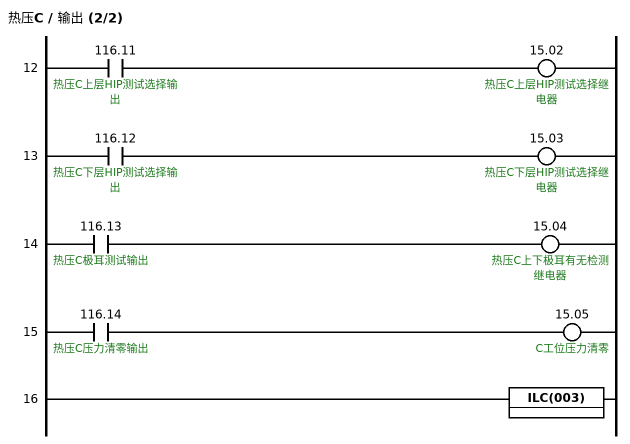
; rung 12
LD 116.11  ; 热压C上层HIP测试选择输出
OUT 15.02  ; 热压C上层HIP测试选择继电器
; rung 13
LD 116.12  ; 热压C下层HIP测试选择输出
OUT 15.03  ; 热压C下层HIP测试选择继电器
; rung 14
LD 116.13  ; 热压C极耳测试输出
OUT 15.04  ; 热压C上下极耳有无检测继电器
; rung 15
LD 116.14  ; 热压C压力清零输出
OUT 15.05  ; C工位压力清零
; rung 16
ILC(003)

### Section END
; rung 0
END(001)

## Program COM (cyclic task 7)

### Section 延时

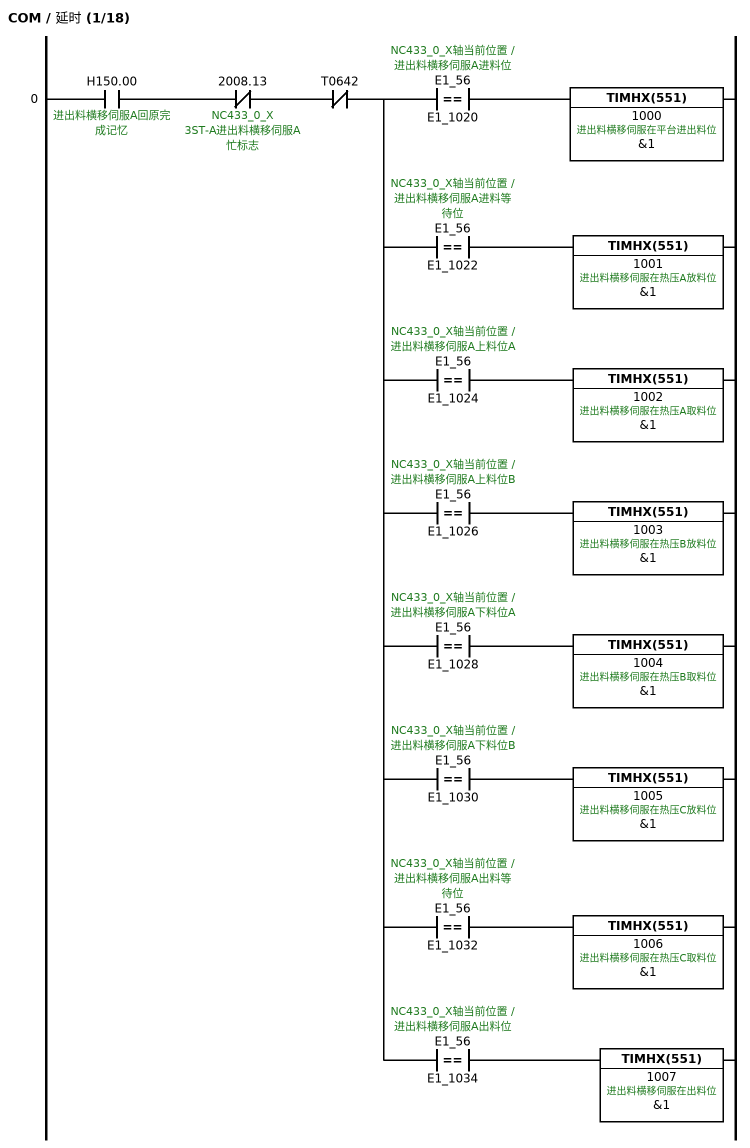
; rung 0
LD H150.00  ; 进出料横移伺服A回原完成记忆
ANDNOT 2008.13  ; NC433_0_X 3ST-A进出料横移伺服A忙标志
ANDNOT T0642
OUT TR0
AND=SL(303) E1_56 E1_1020  ; NC433_0_X轴当前位置, 进出料横移伺服A进料位
TIMHX(551) 1000 &1  ; 进出料横移伺服在平台进出料位
LD TR0
AND=SL(303) E1_56 E1_1022  ; NC433_0_X轴当前位置, 进出料横移伺服A进料等待位
TIMHX(551) 1001 &1  ; 进出料横移伺服在热压A放料位
LD TR0
AND=SL(303) E1_56 E1_1024  ; NC433_0_X轴当前位置, 进出料横移伺服A上料位A
TIMHX(551) 1002 &1  ; 进出料横移伺服在热压A取料位
LD TR0
AND=SL(303) E1_56 E1_1026  ; NC433_0_X轴当前位置, 进出料横移伺服A上料位B
TIMHX(551) 1003 &1  ; 进出料横移伺服在热压B放料位
LD TR0
AND=SL(303) E1_56 E1_1028  ; NC433_0_X轴当前位置, 进出料横移伺服A下料位A
TIMHX(551) 1004 &1  ; 进出料横移伺服在热压B取料位
LD TR0
AND=SL(303) E1_56 E1_1030  ; NC433_0_X轴当前位置, 进出料横移伺服A下料位B
TIMHX(551) 1005 &1  ; 进出料横移伺服在热压C放料位
LD TR0
AND=SL(303) E1_56 E1_1032  ; NC433_0_X轴当前位置, 进出料横移伺服A出料等待位
TIMHX(551) 1006 &1  ; 进出料横移伺服在热压C取料位
LD TR0
AND=SL(303) E1_56 E1_1034  ; NC433_0_X轴当前位置, 进出料横移伺服A出料位
TIMHX(551) 1007 &1  ; 进出料横移伺服在出料位

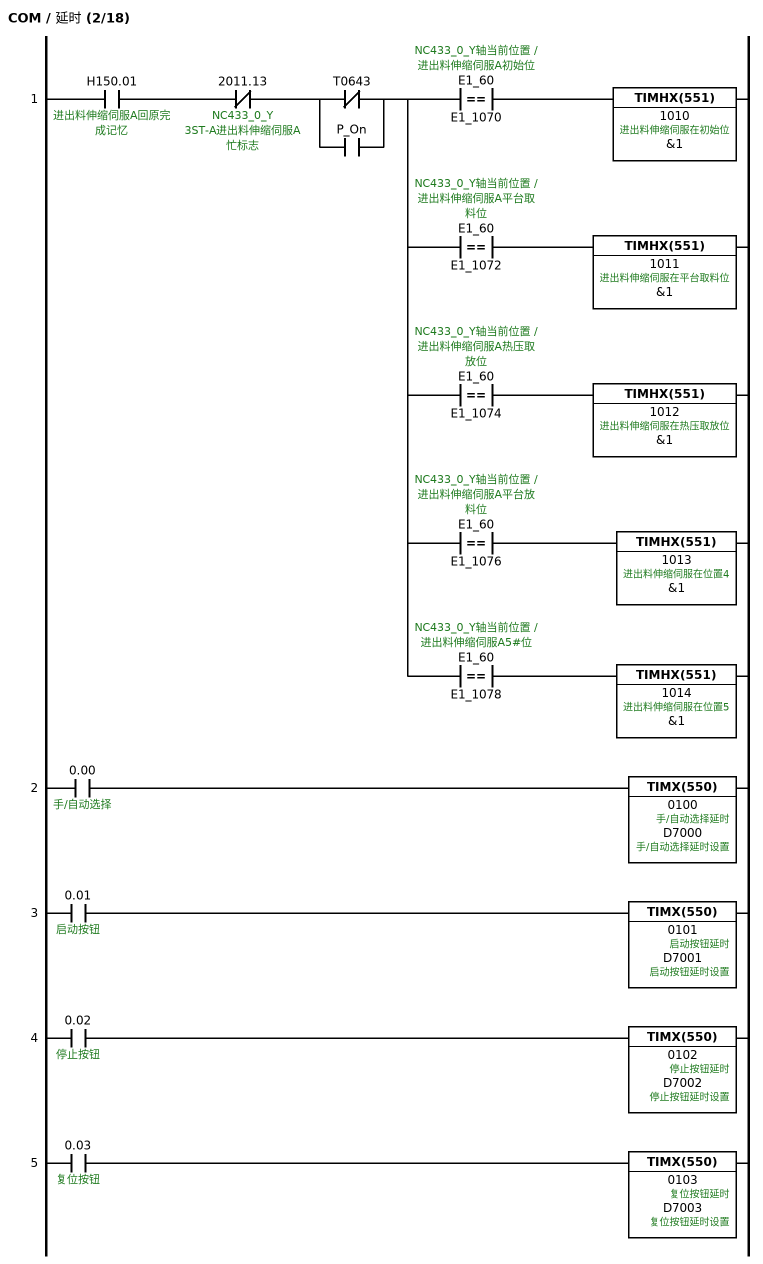
; rung 1
LD H150.01  ; 进出料伸缩伺服A回原完成记忆
ANDNOT 2011.13  ; NC433_0_Y 3ST-A进出料伸缩伺服A忙标志
LDNOT T0643
OR P_On
ANDLD
OUT TR0
AND=SL(303) E1_60 E1_1070  ; NC433_0_Y轴当前位置, 进出料伸缩伺服A初始位
TIMHX(551) 1010 &1  ; 进出料伸缩伺服在初始位
LD TR0
AND=SL(303) E1_60 E1_1072  ; NC433_0_Y轴当前位置, 进出料伸缩伺服A平台取料位
TIMHX(551) 1011 &1  ; 进出料伸缩伺服在平台取料位
LD TR0
AND=SL(303) E1_60 E1_1074  ; NC433_0_Y轴当前位置, 进出料伸缩伺服A热压取放位
TIMHX(551) 1012 &1  ; 进出料伸缩伺服在热压取放位
LD TR0
AND=SL(303) E1_60 E1_1076  ; NC433_0_Y轴当前位置, 进出料伸缩伺服A平台放料位
TIMHX(551) 1013 &1  ; 进出料伸缩伺服在位置4
LD TR0
AND=SL(303) E1_60 E1_1078  ; NC433_0_Y轴当前位置, 进出料伸缩伺服A5#位
TIMHX(551) 1014 &1  ; 进出料伸缩伺服在位置5
; rung 2
LD 0.00  ; 手/自动选择
TIMX(550) 0100 D7000  ; 手/自动选择延时设置, 手/自动选择延时
; rung 3
LD 0.01  ; 启动按钮
TIMX(550) 0101 D7001  ; 启动按钮延时设置, 启动按钮延时
; rung 4
LD 0.02  ; 停止按钮
TIMX(550) 0102 D7002  ; 停止按钮延时设置, 停止按钮延时
; rung 5
LD 0.03  ; 复位按钮
TIMX(550) 0103 D7003  ; 复位按钮延时设置, 复位按钮延时

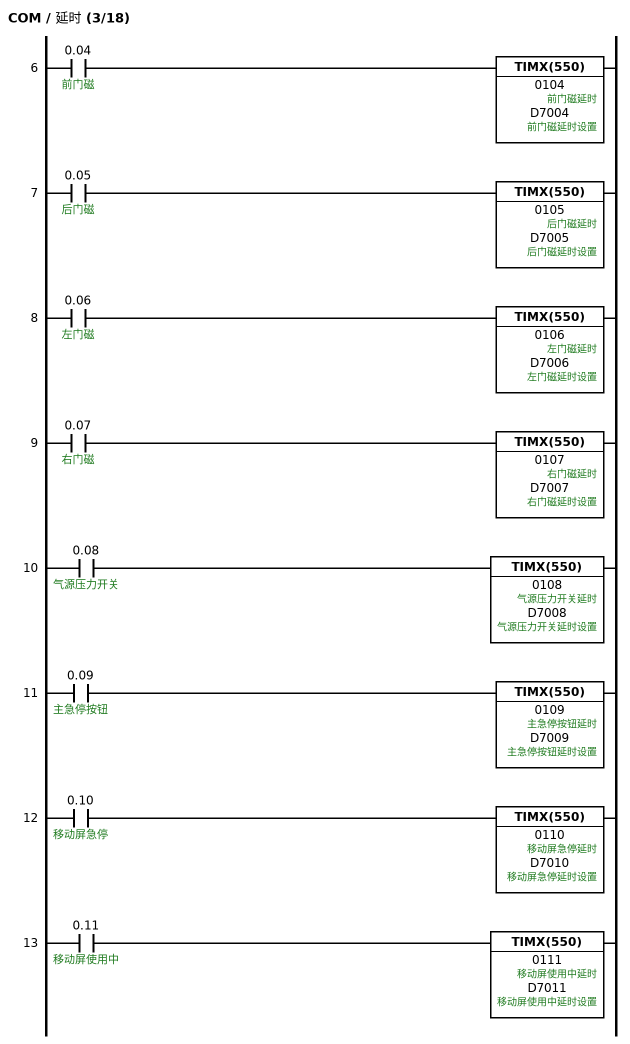
; rung 6
LD 0.04  ; 前门磁
TIMX(550) 0104 D7004  ; 前门磁延时设置, 前门磁延时
; rung 7
LD 0.05  ; 后门磁
TIMX(550) 0105 D7005  ; 后门磁延时设置, 后门磁延时
; rung 8
LD 0.06  ; 左门磁
TIMX(550) 0106 D7006  ; 左门磁延时设置, 左门磁延时
; rung 9
LD 0.07  ; 右门磁
TIMX(550) 0107 D7007  ; 右门磁延时设置, 右门磁延时
; rung 10
LD 0.08  ; 气源压力开关
TIMX(550) 0108 D7008  ; 气源压力开关延时设置, 气源压力开关延时
; rung 11
LD 0.09  ; 主急停按钮
TIMX(550) 0109 D7009  ; 主急停按钮延时设置, 主急停按钮延时
; rung 12
LD 0.10  ; 移动屏急停
TIMX(550) 0110 D7010  ; 移动屏急停延时设置, 移动屏急停延时
; rung 13
LD 0.11  ; 移动屏使用中
TIMX(550) 0111 D7011  ; 移动屏使用中延时设置, 移动屏使用中延时

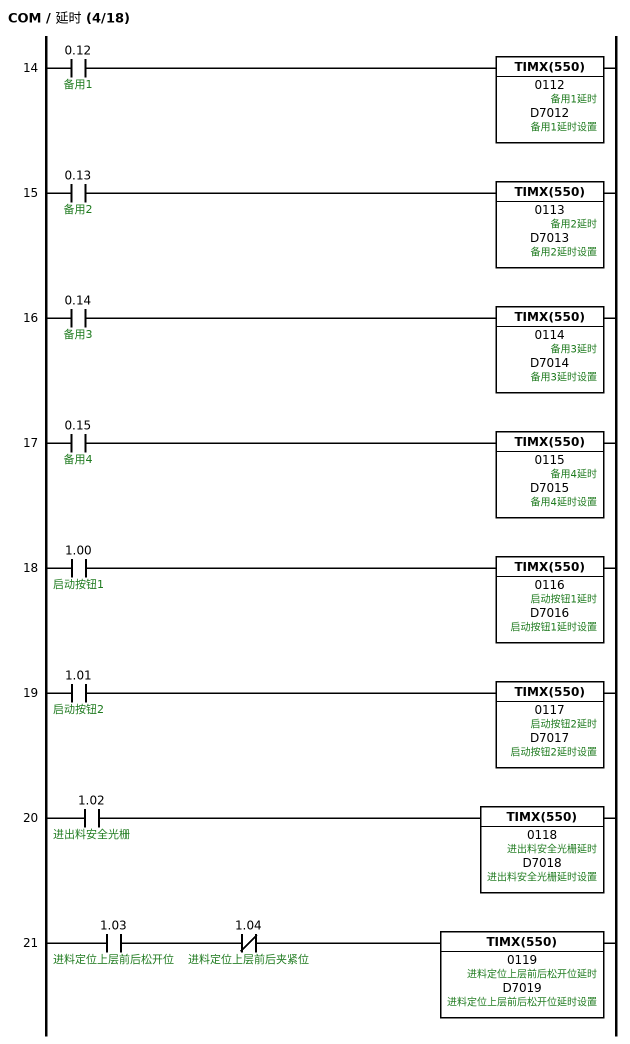
; rung 14
LD 0.12  ; 备用1
TIMX(550) 0112 D7012  ; 备用1延时设置, 备用1延时
; rung 15
LD 0.13  ; 备用2
TIMX(550) 0113 D7013  ; 备用2延时设置, 备用2延时
; rung 16
LD 0.14  ; 备用3
TIMX(550) 0114 D7014  ; 备用3延时设置, 备用3延时
; rung 17
LD 0.15  ; 备用4
TIMX(550) 0115 D7015  ; 备用4延时设置, 备用4延时
; rung 18
LD 1.00  ; 启动按钮1
TIMX(550) 0116 D7016  ; 启动按钮1延时设置, 启动按钮1延时
; rung 19
LD 1.01  ; 启动按钮2
TIMX(550) 0117 D7017  ; 启动按钮2延时设置, 启动按钮2延时
; rung 20
LD 1.02  ; 进出料安全光栅
TIMX(550) 0118 D7018  ; 进出料安全光栅延时设置, 进出料安全光栅延时
; rung 21
LD 1.03  ; 进料定位上层前后松开位
ANDNOT 1.04  ; 进料定位上层前后夹紧位
TIMX(550) 0119 D7019  ; 进料定位上层前后松开位延时设置, 进料定位上层前后松开位延时

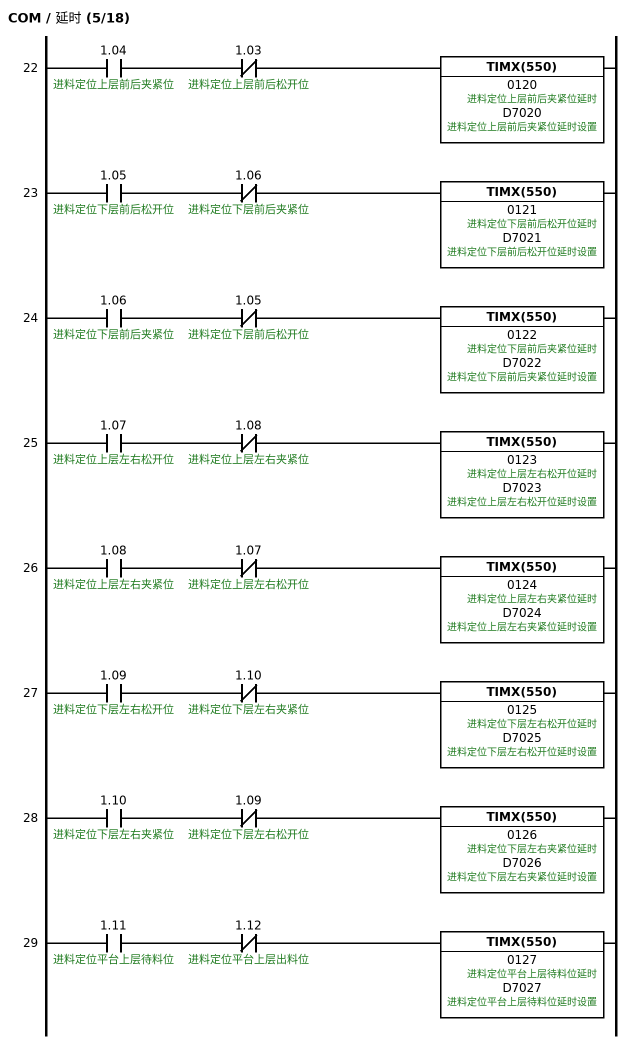
; rung 22
LD 1.04  ; 进料定位上层前后夹紧位
ANDNOT 1.03  ; 进料定位上层前后松开位
TIMX(550) 0120 D7020  ; 进料定位上层前后夹紧位延时设置, 进料定位上层前后夹紧位延时
; rung 23
LD 1.05  ; 进料定位下层前后松开位
ANDNOT 1.06  ; 进料定位下层前后夹紧位
TIMX(550) 0121 D7021  ; 进料定位下层前后松开位延时设置, 进料定位下层前后松开位延时
; rung 24
LD 1.06  ; 进料定位下层前后夹紧位
ANDNOT 1.05  ; 进料定位下层前后松开位
TIMX(550) 0122 D7022  ; 进料定位下层前后夹紧位延时设置, 进料定位下层前后夹紧位延时
; rung 25
LD 1.07  ; 进料定位上层左右松开位
ANDNOT 1.08  ; 进料定位上层左右夹紧位
TIMX(550) 0123 D7023  ; 进料定位上层左右松开位延时设置, 进料定位上层左右松开位延时
; rung 26
LD 1.08  ; 进料定位上层左右夹紧位
ANDNOT 1.07  ; 进料定位上层左右松开位
TIMX(550) 0124 D7024  ; 进料定位上层左右夹紧位延时设置, 进料定位上层左右夹紧位延时
; rung 27
LD 1.09  ; 进料定位下层左右松开位
ANDNOT 1.10  ; 进料定位下层左右夹紧位
TIMX(550) 0125 D7025  ; 进料定位下层左右松开位延时设置, 进料定位下层左右松开位延时
; rung 28
LD 1.10  ; 进料定位下层左右夹紧位
ANDNOT 1.09  ; 进料定位下层左右松开位
TIMX(550) 0126 D7026  ; 进料定位下层左右夹紧位延时设置, 进料定位下层左右夹紧位延时
; rung 29
LD 1.11  ; 进料定位平台上层待料位
ANDNOT 1.12  ; 进料定位平台上层出料位
TIMX(550) 0127 D7027  ; 进料定位平台上层待料位延时设置, 进料定位平台上层待料位延时

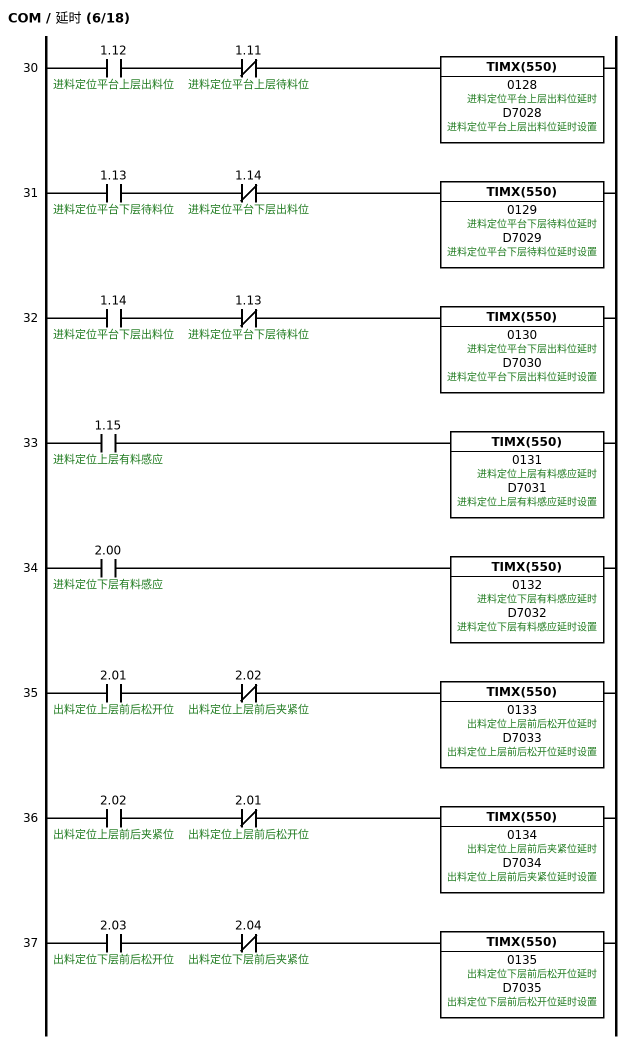
; rung 30
LD 1.12  ; 进料定位平台上层出料位
ANDNOT 1.11  ; 进料定位平台上层待料位
TIMX(550) 0128 D7028  ; 进料定位平台上层出料位延时设置, 进料定位平台上层出料位延时
; rung 31
LD 1.13  ; 进料定位平台下层待料位
ANDNOT 1.14  ; 进料定位平台下层出料位
TIMX(550) 0129 D7029  ; 进料定位平台下层待料位延时设置, 进料定位平台下层待料位延时
; rung 32
LD 1.14  ; 进料定位平台下层出料位
ANDNOT 1.13  ; 进料定位平台下层待料位
TIMX(550) 0130 D7030  ; 进料定位平台下层出料位延时设置, 进料定位平台下层出料位延时
; rung 33
LD 1.15  ; 进料定位上层有料感应
TIMX(550) 0131 D7031  ; 进料定位上层有料感应延时设置, 进料定位上层有料感应延时
; rung 34
LD 2.00  ; 进料定位下层有料感应
TIMX(550) 0132 D7032  ; 进料定位下层有料感应延时设置, 进料定位下层有料感应延时
; rung 35
LD 2.01  ; 出料定位上层前后松开位
ANDNOT 2.02  ; 出料定位上层前后夹紧位
TIMX(550) 0133 D7033  ; 出料定位上层前后松开位延时设置, 出料定位上层前后松开位延时
; rung 36
LD 2.02  ; 出料定位上层前后夹紧位
ANDNOT 2.01  ; 出料定位上层前后松开位
TIMX(550) 0134 D7034  ; 出料定位上层前后夹紧位延时设置, 出料定位上层前后夹紧位延时
; rung 37
LD 2.03  ; 出料定位下层前后松开位
ANDNOT 2.04  ; 出料定位下层前后夹紧位
TIMX(550) 0135 D7035  ; 出料定位下层前后松开位延时设置, 出料定位下层前后松开位延时

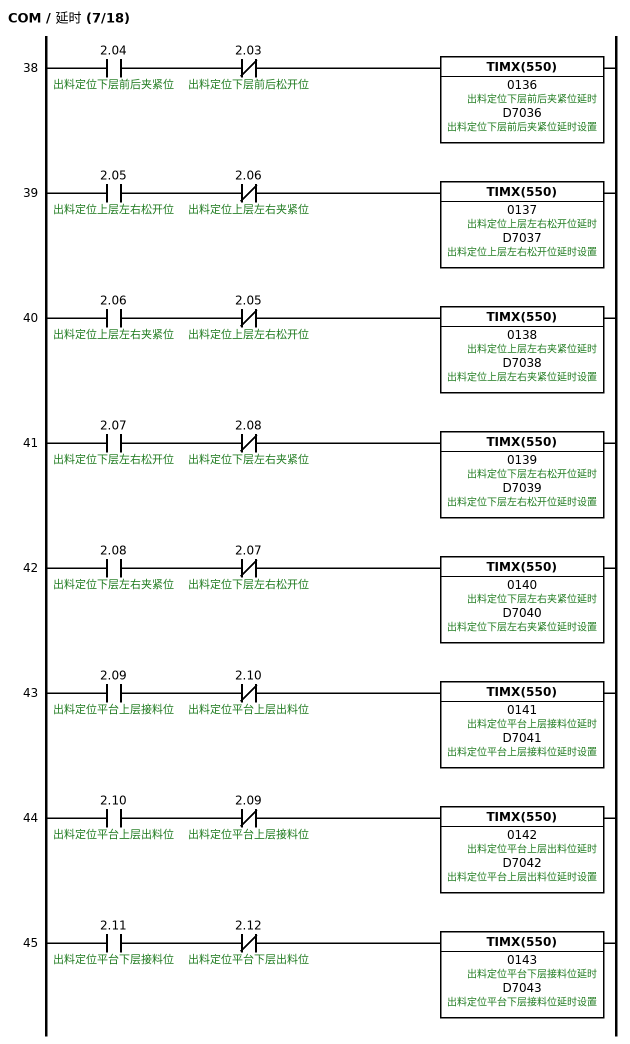
; rung 38
LD 2.04  ; 出料定位下层前后夹紧位
ANDNOT 2.03  ; 出料定位下层前后松开位
TIMX(550) 0136 D7036  ; 出料定位下层前后夹紧位延时设置, 出料定位下层前后夹紧位延时
; rung 39
LD 2.05  ; 出料定位上层左右松开位
ANDNOT 2.06  ; 出料定位上层左右夹紧位
TIMX(550) 0137 D7037  ; 出料定位上层左右松开位延时设置, 出料定位上层左右松开位延时
; rung 40
LD 2.06  ; 出料定位上层左右夹紧位
ANDNOT 2.05  ; 出料定位上层左右松开位
TIMX(550) 0138 D7038  ; 出料定位上层左右夹紧位延时设置, 出料定位上层左右夹紧位延时
; rung 41
LD 2.07  ; 出料定位下层左右松开位
ANDNOT 2.08  ; 出料定位下层左右夹紧位
TIMX(550) 0139 D7039  ; 出料定位下层左右松开位延时设置, 出料定位下层左右松开位延时
; rung 42
LD 2.08  ; 出料定位下层左右夹紧位
ANDNOT 2.07  ; 出料定位下层左右松开位
TIMX(550) 0140 D7040  ; 出料定位下层左右夹紧位延时设置, 出料定位下层左右夹紧位延时
; rung 43
LD 2.09  ; 出料定位平台上层接料位
ANDNOT 2.10  ; 出料定位平台上层出料位
TIMX(550) 0141 D7041  ; 出料定位平台上层接料位延时设置, 出料定位平台上层接料位延时
; rung 44
LD 2.10  ; 出料定位平台上层出料位
ANDNOT 2.09  ; 出料定位平台上层接料位
TIMX(550) 0142 D7042  ; 出料定位平台上层出料位延时设置, 出料定位平台上层出料位延时
; rung 45
LD 2.11  ; 出料定位平台下层接料位
ANDNOT 2.12  ; 出料定位平台下层出料位
TIMX(550) 0143 D7043  ; 出料定位平台下层接料位延时设置, 出料定位平台下层接料位延时

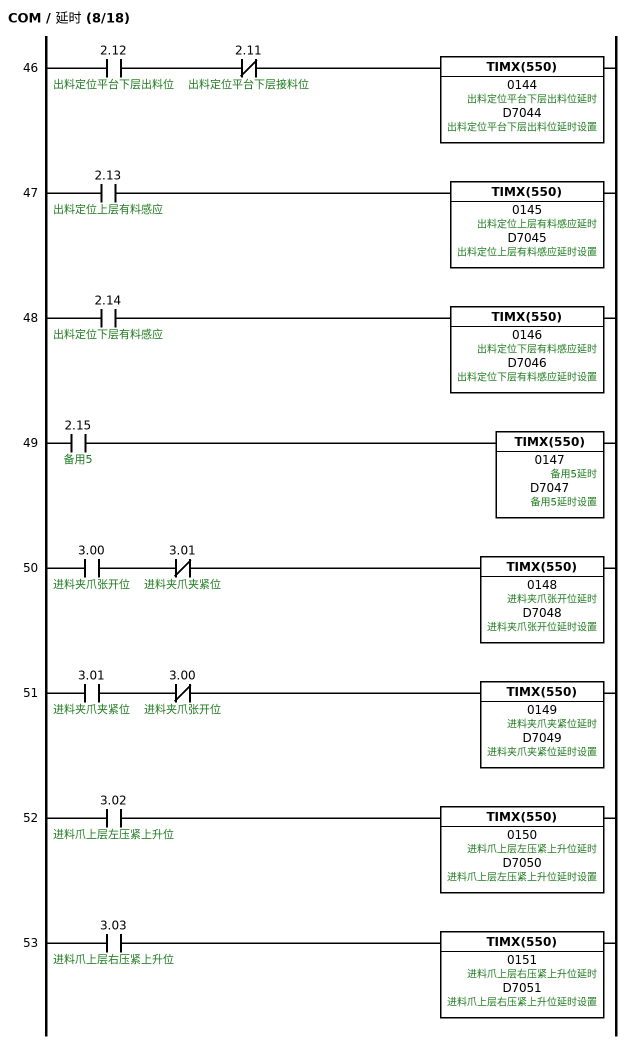
; rung 46
LD 2.12  ; 出料定位平台下层出料位
ANDNOT 2.11  ; 出料定位平台下层接料位
TIMX(550) 0144 D7044  ; 出料定位平台下层出料位延时设置, 出料定位平台下层出料位延时
; rung 47
LD 2.13  ; 出料定位上层有料感应
TIMX(550) 0145 D7045  ; 出料定位上层有料感应延时设置, 出料定位上层有料感应延时
; rung 48
LD 2.14  ; 出料定位下层有料感应
TIMX(550) 0146 D7046  ; 出料定位下层有料感应延时设置, 出料定位下层有料感应延时
; rung 49
LD 2.15  ; 备用5
TIMX(550) 0147 D7047  ; 备用5延时设置, 备用5延时
; rung 50
LD 3.00  ; 进料夹爪张开位
ANDNOT 3.01  ; 进料夹爪夹紧位
TIMX(550) 0148 D7048  ; 进料夹爪张开位延时设置, 进料夹爪张开位延时
; rung 51
LD 3.01  ; 进料夹爪夹紧位
ANDNOT 3.00  ; 进料夹爪张开位
TIMX(550) 0149 D7049  ; 进料夹爪夹紧位延时设置, 进料夹爪夹紧位延时
; rung 52
LD 3.02  ; 进料爪上层左压紧上升位
TIMX(550) 0150 D7050  ; 进料爪上层左压紧上升位延时设置, 进料爪上层左压紧上升位延时
; rung 53
LD 3.03  ; 进料爪上层右压紧上升位
TIMX(550) 0151 D7051  ; 进料爪上层右压紧上升位延时设置, 进料爪上层右压紧上升位延时

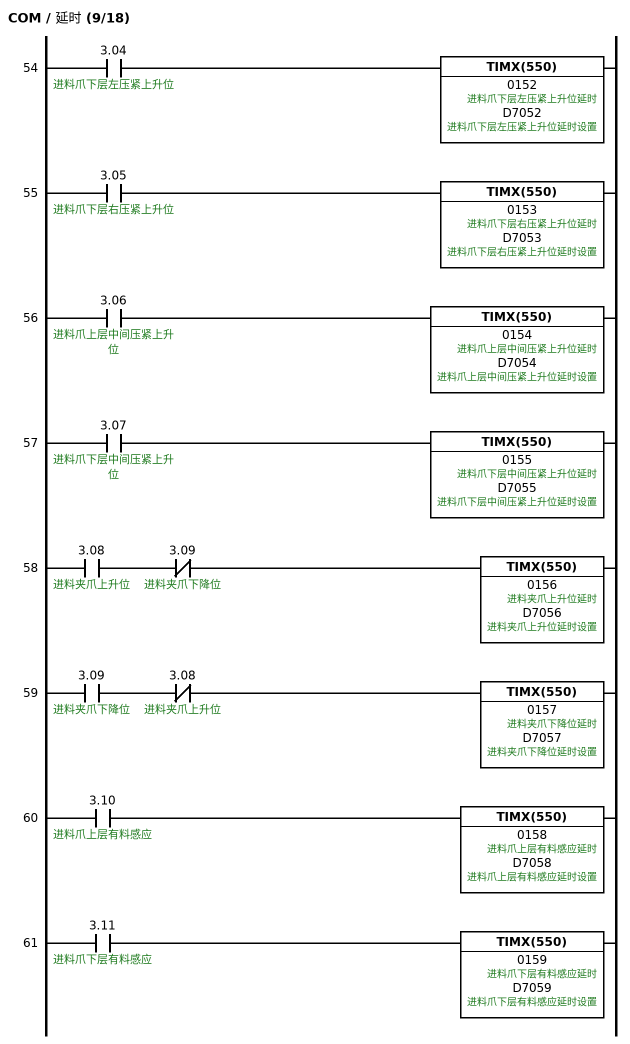
; rung 54
LD 3.04  ; 进料爪下层左压紧上升位
TIMX(550) 0152 D7052  ; 进料爪下层左压紧上升位延时设置, 进料爪下层左压紧上升位延时
; rung 55
LD 3.05  ; 进料爪下层右压紧上升位
TIMX(550) 0153 D7053  ; 进料爪下层右压紧上升位延时设置, 进料爪下层右压紧上升位延时
; rung 56
LD 3.06  ; 进料爪上层中间压紧上升位
TIMX(550) 0154 D7054  ; 进料爪上层中间压紧上升位延时设置, 进料爪上层中间压紧上升位延时
; rung 57
LD 3.07  ; 进料爪下层中间压紧上升位
TIMX(550) 0155 D7055  ; 进料爪下层中间压紧上升位延时设置, 进料爪下层中间压紧上升位延时
; rung 58
LD 3.08  ; 进料夹爪上升位
ANDNOT 3.09  ; 进料夹爪下降位
TIMX(550) 0156 D7056  ; 进料夹爪上升位延时设置, 进料夹爪上升位延时
; rung 59
LD 3.09  ; 进料夹爪下降位
ANDNOT 3.08  ; 进料夹爪上升位
TIMX(550) 0157 D7057  ; 进料夹爪下降位延时设置, 进料夹爪下降位延时
; rung 60
LD 3.10  ; 进料爪上层有料感应
TIMX(550) 0158 D7058  ; 进料爪上层有料感应延时设置, 进料爪上层有料感应延时
; rung 61
LD 3.11  ; 进料爪下层有料感应
TIMX(550) 0159 D7059  ; 进料爪下层有料感应延时设置, 进料爪下层有料感应延时

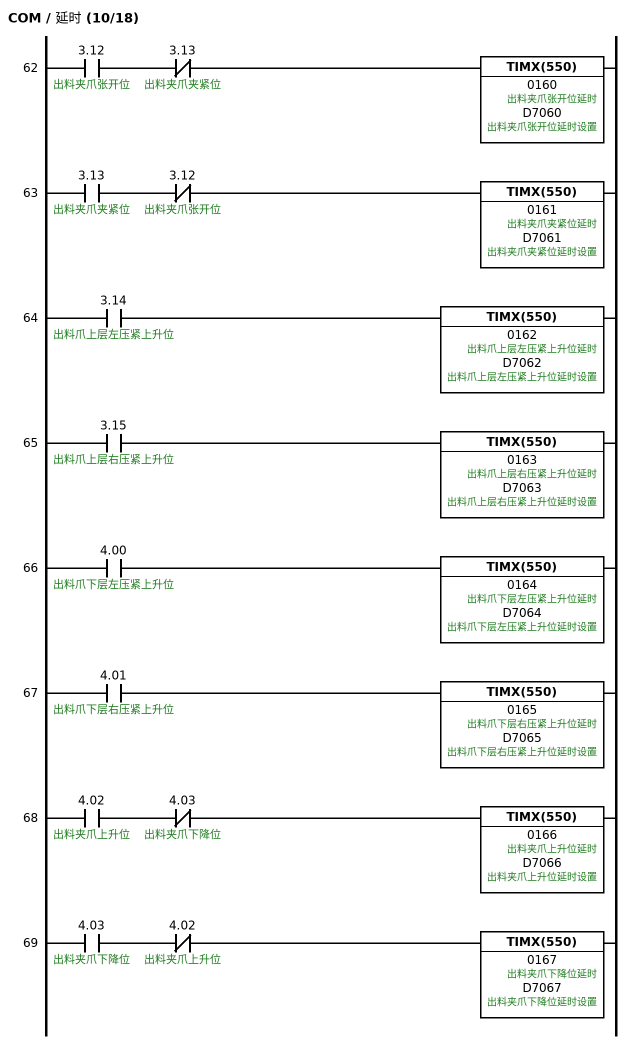
; rung 62
LD 3.12  ; 出料夹爪张开位
ANDNOT 3.13  ; 出料夹爪夹紧位
TIMX(550) 0160 D7060  ; 出料夹爪张开位延时设置, 出料夹爪张开位延时
; rung 63
LD 3.13  ; 出料夹爪夹紧位
ANDNOT 3.12  ; 出料夹爪张开位
TIMX(550) 0161 D7061  ; 出料夹爪夹紧位延时设置, 出料夹爪夹紧位延时
; rung 64
LD 3.14  ; 出料爪上层左压紧上升位
TIMX(550) 0162 D7062  ; 出料爪上层左压紧上升位延时设置, 出料爪上层左压紧上升位延时
; rung 65
LD 3.15  ; 出料爪上层右压紧上升位
TIMX(550) 0163 D7063  ; 出料爪上层右压紧上升位延时设置, 出料爪上层右压紧上升位延时
; rung 66
LD 4.00  ; 出料爪下层左压紧上升位
TIMX(550) 0164 D7064  ; 出料爪下层左压紧上升位延时设置, 出料爪下层左压紧上升位延时
; rung 67
LD 4.01  ; 出料爪下层右压紧上升位
TIMX(550) 0165 D7065  ; 出料爪下层右压紧上升位延时设置, 出料爪下层右压紧上升位延时
; rung 68
LD 4.02  ; 出料夹爪上升位
ANDNOT 4.03  ; 出料夹爪下降位
TIMX(550) 0166 D7066  ; 出料夹爪上升位延时设置, 出料夹爪上升位延时
; rung 69
LD 4.03  ; 出料夹爪下降位
ANDNOT 4.02  ; 出料夹爪上升位
TIMX(550) 0167 D7067  ; 出料夹爪下降位延时设置, 出料夹爪下降位延时

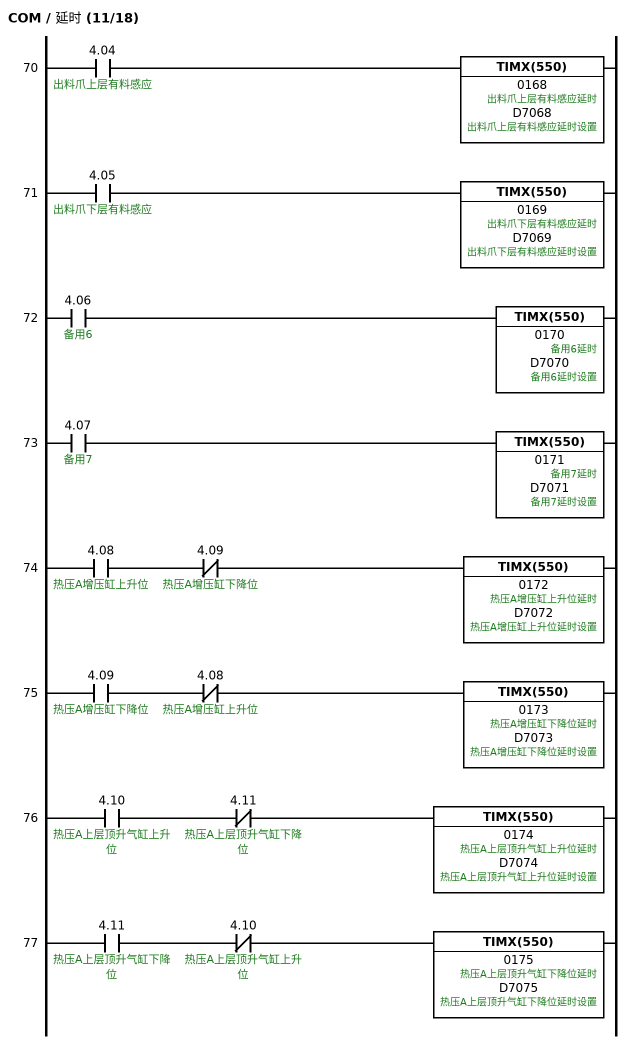
; rung 70
LD 4.04  ; 出料爪上层有料感应
TIMX(550) 0168 D7068  ; 出料爪上层有料感应延时设置, 出料爪上层有料感应延时
; rung 71
LD 4.05  ; 出料爪下层有料感应
TIMX(550) 0169 D7069  ; 出料爪下层有料感应延时设置, 出料爪下层有料感应延时
; rung 72
LD 4.06  ; 备用6
TIMX(550) 0170 D7070  ; 备用6延时设置, 备用6延时
; rung 73
LD 4.07  ; 备用7
TIMX(550) 0171 D7071  ; 备用7延时设置, 备用7延时
; rung 74
LD 4.08  ; 热压A增压缸上升位
ANDNOT 4.09  ; 热压A增压缸下降位
TIMX(550) 0172 D7072  ; 热压A增压缸上升位延时设置, 热压A增压缸上升位延时
; rung 75
LD 4.09  ; 热压A增压缸下降位
ANDNOT 4.08  ; 热压A增压缸上升位
TIMX(550) 0173 D7073  ; 热压A增压缸下降位延时设置, 热压A增压缸下降位延时
; rung 76
LD 4.10  ; 热压A上层顶升气缸上升位
ANDNOT 4.11  ; 热压A上层顶升气缸下降位
TIMX(550) 0174 D7074  ; 热压A上层顶升气缸上升位延时设置, 热压A上层顶升气缸上升位延时
; rung 77
LD 4.11  ; 热压A上层顶升气缸下降位
ANDNOT 4.10  ; 热压A上层顶升气缸上升位
TIMX(550) 0175 D7075  ; 热压A上层顶升气缸下降位延时设置, 热压A上层顶升气缸下降位延时

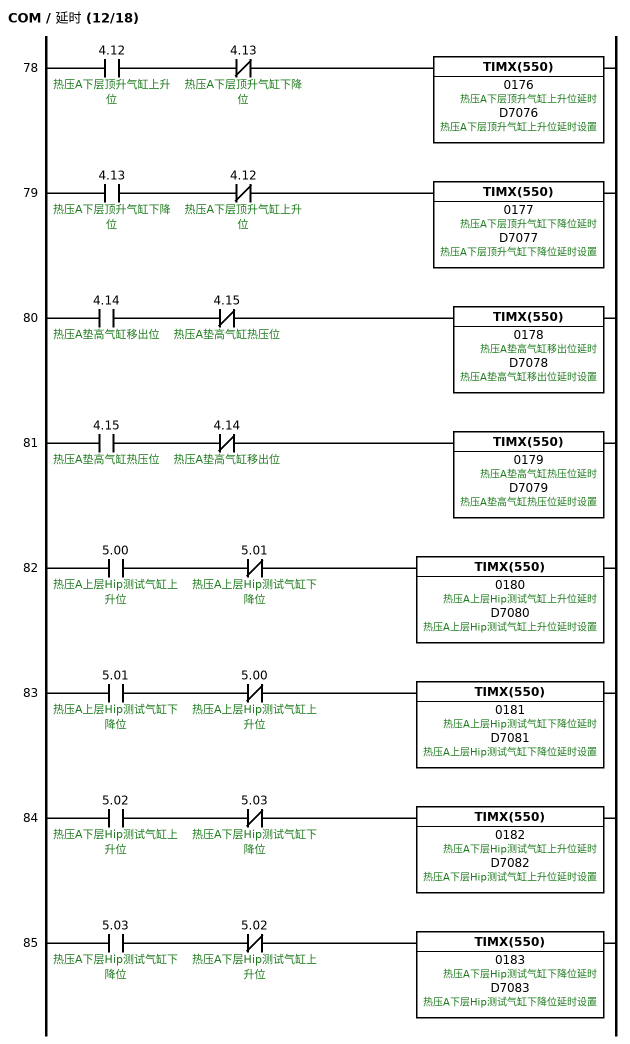
; rung 78
LD 4.12  ; 热压A下层顶升气缸上升位
ANDNOT 4.13  ; 热压A下层顶升气缸下降位
TIMX(550) 0176 D7076  ; 热压A下层顶升气缸上升位延时设置, 热压A下层顶升气缸上升位延时
; rung 79
LD 4.13  ; 热压A下层顶升气缸下降位
ANDNOT 4.12  ; 热压A下层顶升气缸上升位
TIMX(550) 0177 D7077  ; 热压A下层顶升气缸下降位延时设置, 热压A下层顶升气缸下降位延时
; rung 80
LD 4.14  ; 热压A垫高气缸移出位
ANDNOT 4.15  ; 热压A垫高气缸热压位
TIMX(550) 0178 D7078  ; 热压A垫高气缸移出位延时设置, 热压A垫高气缸移出位延时
; rung 81
LD 4.15  ; 热压A垫高气缸热压位
ANDNOT 4.14  ; 热压A垫高气缸移出位
TIMX(550) 0179 D7079  ; 热压A垫高气缸热压位延时设置, 热压A垫高气缸热压位延时
; rung 82
LD 5.00  ; 热压A上层Hip测试气缸上升位
ANDNOT 5.01  ; 热压A上层Hip测试气缸下降位
TIMX(550) 0180 D7080  ; 热压A上层Hip测试气缸上升位延时设置, 热压A上层Hip测试气缸上升位延时
; rung 83
LD 5.01  ; 热压A上层Hip测试气缸下降位
ANDNOT 5.00  ; 热压A上层Hip测试气缸上升位
TIMX(550) 0181 D7081  ; 热压A上层Hip测试气缸下降位延时设置, 热压A上层Hip测试气缸下降位延时
; rung 84
LD 5.02  ; 热压A下层Hip测试气缸上升位
ANDNOT 5.03  ; 热压A下层Hip测试气缸下降位
TIMX(550) 0182 D7082  ; 热压A下层Hip测试气缸上升位延时设置, 热压A下层Hip测试气缸上升位延时
; rung 85
LD 5.03  ; 热压A下层Hip测试气缸下降位
ANDNOT 5.02  ; 热压A下层Hip测试气缸上升位
TIMX(550) 0183 D7083  ; 热压A下层Hip测试气缸下降位延时设置, 热压A下层Hip测试气缸下降位延时

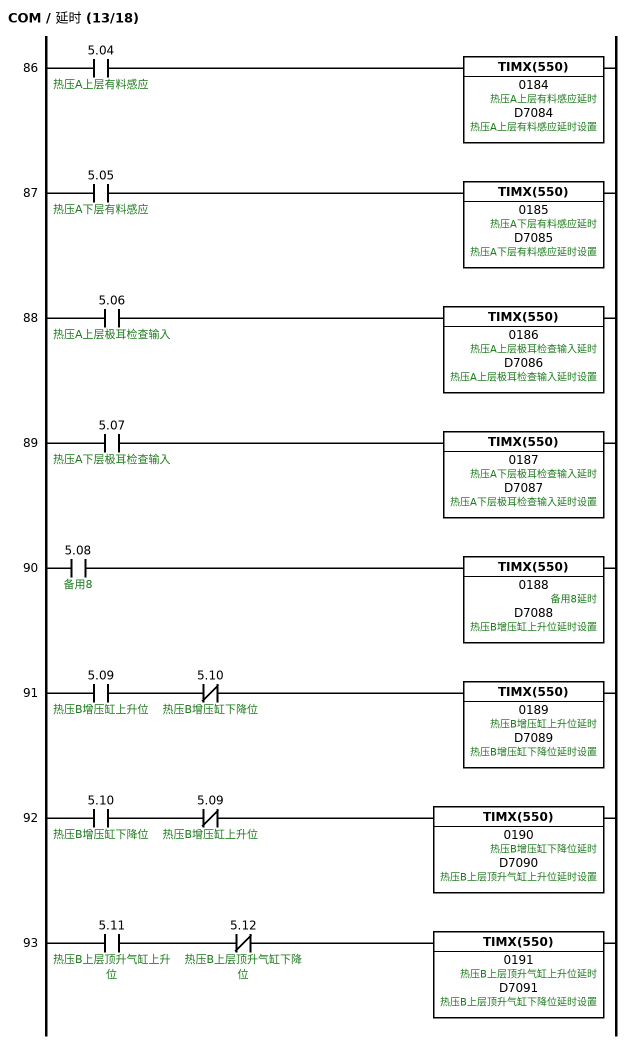
; rung 86
LD 5.04  ; 热压A上层有料感应
TIMX(550) 0184 D7084  ; 热压A上层有料感应延时设置, 热压A上层有料感应延时
; rung 87
LD 5.05  ; 热压A下层有料感应
TIMX(550) 0185 D7085  ; 热压A下层有料感应延时设置, 热压A下层有料感应延时
; rung 88
LD 5.06  ; 热压A上层极耳检查输入
TIMX(550) 0186 D7086  ; 热压A上层极耳检查输入延时设置, 热压A上层极耳检查输入延时
; rung 89
LD 5.07  ; 热压A下层极耳检查输入
TIMX(550) 0187 D7087  ; 热压A下层极耳检查输入延时设置, 热压A下层极耳检查输入延时
; rung 90
LD 5.08  ; 备用8
TIMX(550) 0188 D7088  ; 热压B增压缸上升位延时设置, 备用8延时
; rung 91
LD 5.09  ; 热压B增压缸上升位
ANDNOT 5.10  ; 热压B增压缸下降位
TIMX(550) 0189 D7089  ; 热压B增压缸下降位延时设置, 热压B增压缸上升位延时
; rung 92
LD 5.10  ; 热压B增压缸下降位
ANDNOT 5.09  ; 热压B增压缸上升位
TIMX(550) 0190 D7090  ; 热压B上层顶升气缸上升位延时设置, 热压B增压缸下降位延时
; rung 93
LD 5.11  ; 热压B上层顶升气缸上升位
ANDNOT 5.12  ; 热压B上层顶升气缸下降位
TIMX(550) 0191 D7091  ; 热压B上层顶升气缸下降位延时设置, 热压B上层顶升气缸上升位延时

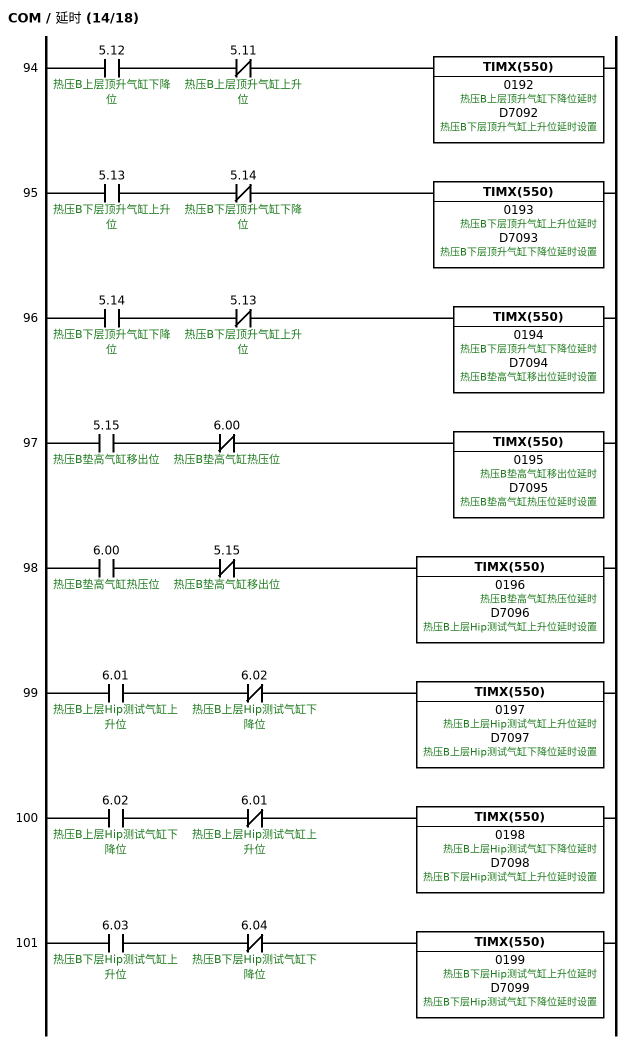
; rung 94
LD 5.12  ; 热压B上层顶升气缸下降位
ANDNOT 5.11  ; 热压B上层顶升气缸上升位
TIMX(550) 0192 D7092  ; 热压B下层顶升气缸上升位延时设置, 热压B上层顶升气缸下降位延时
; rung 95
LD 5.13  ; 热压B下层顶升气缸上升位
ANDNOT 5.14  ; 热压B下层顶升气缸下降位
TIMX(550) 0193 D7093  ; 热压B下层顶升气缸下降位延时设置, 热压B下层顶升气缸上升位延时
; rung 96
LD 5.14  ; 热压B下层顶升气缸下降位
ANDNOT 5.13  ; 热压B下层顶升气缸上升位
TIMX(550) 0194 D7094  ; 热压B垫高气缸移出位延时设置, 热压B下层顶升气缸下降位延时
; rung 97
LD 5.15  ; 热压B垫高气缸移出位
ANDNOT 6.00  ; 热压B垫高气缸热压位
TIMX(550) 0195 D7095  ; 热压B垫高气缸热压位延时设置, 热压B垫高气缸移出位延时
; rung 98
LD 6.00  ; 热压B垫高气缸热压位
ANDNOT 5.15  ; 热压B垫高气缸移出位
TIMX(550) 0196 D7096  ; 热压B上层Hip测试气缸上升位延时设置, 热压B垫高气缸热压位延时
; rung 99
LD 6.01  ; 热压B上层Hip测试气缸上升位
ANDNOT 6.02  ; 热压B上层Hip测试气缸下降位
TIMX(550) 0197 D7097  ; 热压B上层Hip测试气缸下降位延时设置, 热压B上层Hip测试气缸上升位延时
; rung 100
LD 6.02  ; 热压B上层Hip测试气缸下降位
ANDNOT 6.01  ; 热压B上层Hip测试气缸上升位
TIMX(550) 0198 D7098  ; 热压B下层Hip测试气缸上升位延时设置, 热压B上层Hip测试气缸下降位延时
; rung 101
LD 6.03  ; 热压B下层Hip测试气缸上升位
ANDNOT 6.04  ; 热压B下层Hip测试气缸下降位
TIMX(550) 0199 D7099  ; 热压B下层Hip测试气缸下降位延时设置, 热压B下层Hip测试气缸上升位延时

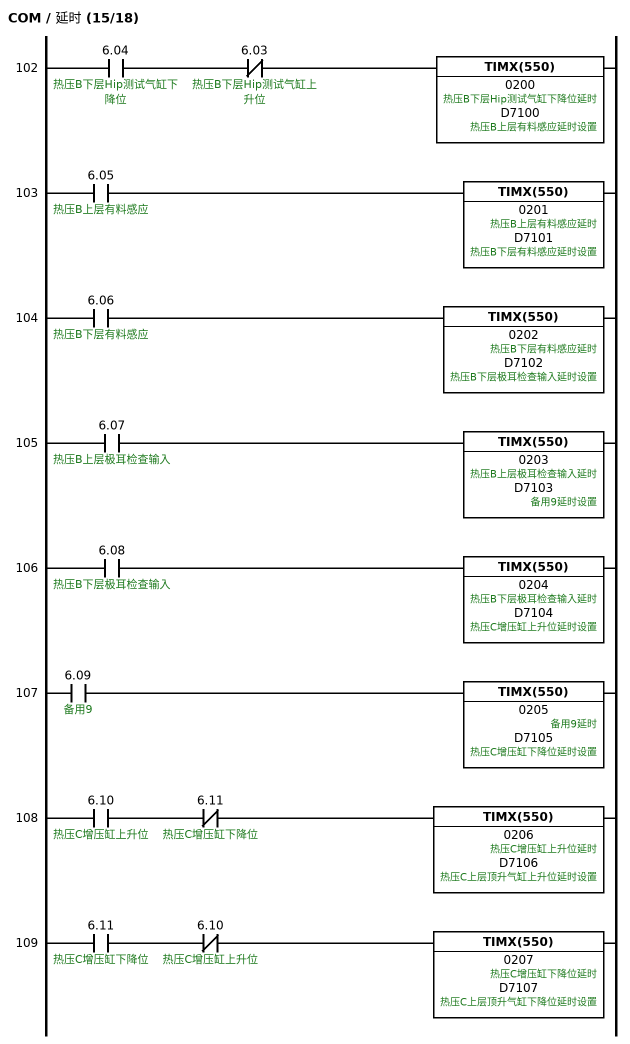
; rung 102
LD 6.04  ; 热压B下层Hip测试气缸下降位
ANDNOT 6.03  ; 热压B下层Hip测试气缸上升位
TIMX(550) 0200 D7100  ; 热压B上层有料感应延时设置, 热压B下层Hip测试气缸下降位延时
; rung 103
LD 6.05  ; 热压B上层有料感应
TIMX(550) 0201 D7101  ; 热压B下层有料感应延时设置, 热压B上层有料感应延时
; rung 104
LD 6.06  ; 热压B下层有料感应
TIMX(550) 0202 D7102  ; 热压B下层极耳检查输入延时设置, 热压B下层有料感应延时
; rung 105
LD 6.07  ; 热压B上层极耳检查输入
TIMX(550) 0203 D7103  ; 备用9延时设置, 热压B上层极耳检查输入延时
; rung 106
LD 6.08  ; 热压B下层极耳检查输入
TIMX(550) 0204 D7104  ; 热压C增压缸上升位延时设置, 热压B下层极耳检查输入延时
; rung 107
LD 6.09  ; 备用9
TIMX(550) 0205 D7105  ; 热压C增压缸下降位延时设置, 备用9延时
; rung 108
LD 6.10  ; 热压C增压缸上升位
ANDNOT 6.11  ; 热压C增压缸下降位
TIMX(550) 0206 D7106  ; 热压C上层顶升气缸上升位延时设置, 热压C增压缸上升位延时
; rung 109
LD 6.11  ; 热压C增压缸下降位
ANDNOT 6.10  ; 热压C增压缸上升位
TIMX(550) 0207 D7107  ; 热压C上层顶升气缸下降位延时设置, 热压C增压缸下降位延时

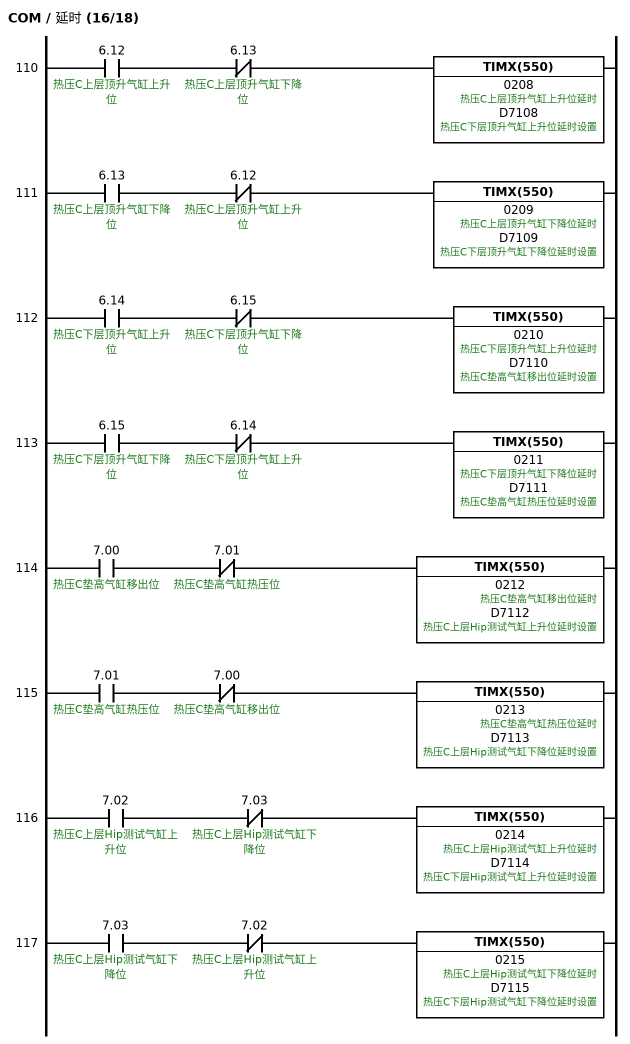
; rung 110
LD 6.12  ; 热压C上层顶升气缸上升位
ANDNOT 6.13  ; 热压C上层顶升气缸下降位
TIMX(550) 0208 D7108  ; 热压C下层顶升气缸上升位延时设置, 热压C上层顶升气缸上升位延时
; rung 111
LD 6.13  ; 热压C上层顶升气缸下降位
ANDNOT 6.12  ; 热压C上层顶升气缸上升位
TIMX(550) 0209 D7109  ; 热压C下层顶升气缸下降位延时设置, 热压C上层顶升气缸下降位延时
; rung 112
LD 6.14  ; 热压C下层顶升气缸上升位
ANDNOT 6.15  ; 热压C下层顶升气缸下降位
TIMX(550) 0210 D7110  ; 热压C垫高气缸移出位延时设置, 热压C下层顶升气缸上升位延时
; rung 113
LD 6.15  ; 热压C下层顶升气缸下降位
ANDNOT 6.14  ; 热压C下层顶升气缸上升位
TIMX(550) 0211 D7111  ; 热压C垫高气缸热压位延时设置, 热压C下层顶升气缸下降位延时
; rung 114
LD 7.00  ; 热压C垫高气缸移出位
ANDNOT 7.01  ; 热压C垫高气缸热压位
TIMX(550) 0212 D7112  ; 热压C上层Hip测试气缸上升位延时设置, 热压C垫高气缸移出位延时
; rung 115
LD 7.01  ; 热压C垫高气缸热压位
ANDNOT 7.00  ; 热压C垫高气缸移出位
TIMX(550) 0213 D7113  ; 热压C上层Hip测试气缸下降位延时设置, 热压C垫高气缸热压位延时
; rung 116
LD 7.02  ; 热压C上层Hip测试气缸上升位
ANDNOT 7.03  ; 热压C上层Hip测试气缸下降位
TIMX(550) 0214 D7114  ; 热压C下层Hip测试气缸上升位延时设置, 热压C上层Hip测试气缸上升位延时
; rung 117
LD 7.03  ; 热压C上层Hip测试气缸下降位
ANDNOT 7.02  ; 热压C上层Hip测试气缸上升位
TIMX(550) 0215 D7115  ; 热压C下层Hip测试气缸下降位延时设置, 热压C上层Hip测试气缸下降位延时

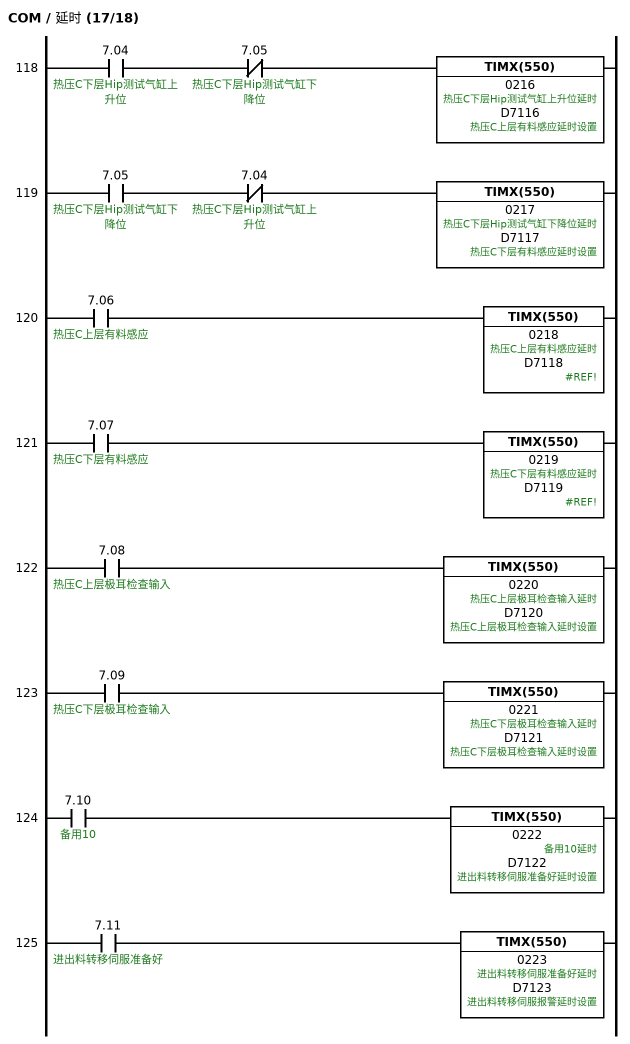
; rung 118
LD 7.04  ; 热压C下层Hip测试气缸上升位
ANDNOT 7.05  ; 热压C下层Hip测试气缸下降位
TIMX(550) 0216 D7116  ; 热压C上层有料感应延时设置, 热压C下层Hip测试气缸上升位延时
; rung 119
LD 7.05  ; 热压C下层Hip测试气缸下降位
ANDNOT 7.04  ; 热压C下层Hip测试气缸上升位
TIMX(550) 0217 D7117  ; 热压C下层有料感应延时设置, 热压C下层Hip测试气缸下降位延时
; rung 120
LD 7.06  ; 热压C上层有料感应
TIMX(550) 0218 D7118  ; #REF!, 热压C上层有料感应延时
; rung 121
LD 7.07  ; 热压C下层有料感应
TIMX(550) 0219 D7119  ; #REF!, 热压C下层有料感应延时
; rung 122
LD 7.08  ; 热压C上层极耳检查输入
TIMX(550) 0220 D7120  ; 热压C上层极耳检查输入延时设置, 热压C上层极耳检查输入延时
; rung 123
LD 7.09  ; 热压C下层极耳检查输入
TIMX(550) 0221 D7121  ; 热压C下层极耳检查输入延时设置, 热压C下层极耳检查输入延时
; rung 124
LD 7.10  ; 备用10
TIMX(550) 0222 D7122  ; 进出料转移伺服准备好延时设置, 备用10延时
; rung 125
LD 7.11  ; 进出料转移伺服准备好
TIMX(550) 0223 D7123  ; 进出料转移伺服报警延时设置, 进出料转移伺服准备好延时

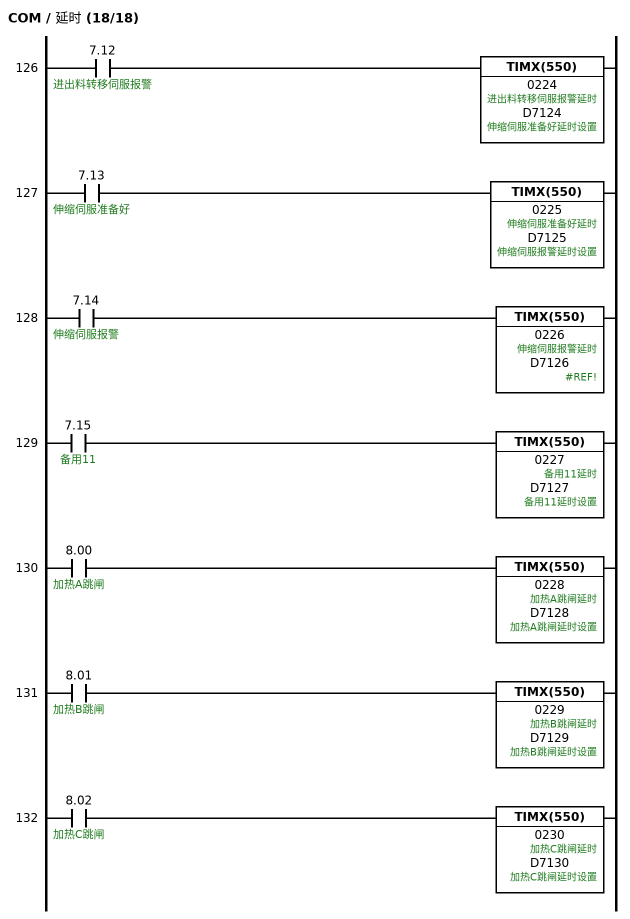
; rung 126
LD 7.12  ; 进出料转移伺服报警
TIMX(550) 0224 D7124  ; 伸缩伺服准备好延时设置, 进出料转移伺服报警延时
; rung 127
LD 7.13  ; 伸缩伺服准备好
TIMX(550) 0225 D7125  ; 伸缩伺服报警延时设置, 伸缩伺服准备好延时
; rung 128
LD 7.14  ; 伸缩伺服报警
TIMX(550) 0226 D7126  ; #REF!, 伸缩伺服报警延时
; rung 129
LD 7.15  ; 备用11
TIMX(550) 0227 D7127  ; 备用11延时设置, 备用11延时
; rung 130
LD 8.00  ; 加热A跳闸
TIMX(550) 0228 D7128  ; 加热A跳闸延时设置, 加热A跳闸延时
; rung 131
LD 8.01  ; 加热B跳闸
TIMX(550) 0229 D7129  ; 加热B跳闸延时设置, 加热B跳闸延时
; rung 132
LD 8.02  ; 加热C跳闸
TIMX(550) 0230 D7130  ; 加热C跳闸延时设置, 加热C跳闸延时

### Section END
; rung 0
END(001)

## Function block _NCx011A_MoveAbsolute_DINT (Omron library block, body left out)

## Function block _NCx021_MoveRelative_DINT (Omron library block, body left out)

## Function block _NCx051A_Home_DINT (Omron library block, body left out)

## Function block _NCx600_Setting (Omron library block, body left out)

## Function block H_Pit_Read_Resistance_Value
VAR_INPUT
  启动测试 : BOOL;
  NOCOMP比较停用 : BOOL;  (* $?St$Bk?_#[578] / "NOCOMP"结果比较停用$?St$Bk?_#[578] *)
  Hipot复测启用 : BOOL;  (* Hipot复测启用 *)
  通讯异常复位 : BOOL;  (* ST5520_Hipot通讯异常复位 *)
  端口控制字 : WORD;
  启动控制字 : WORD;
  通讯端口忙标志 : BOOL;
  读取电阻控制字 : WORD;
  读取电压控制字 : WORD;
  测试时间 : UINT;  (* 延时读取绝缘仪测试值时间 *)
  复测次数 : UINT;  (* 设置复测次数 *)
  INT1 : UINT;
END_VAR
VAR_OUTPUT
  绝缘测试值 : REAL;  (* ST5520_返回绝缘测试兆欧值(Float) *)
  NG类型 : REAL;  (* ST5520_测试结果(位) *)
  测试结果 : REAL;  (* ST5520_测试结果(字) *)
  测试实时电压 : REAL;
  测试完成 : BOOL;
  通讯异常 : BOOL;  (* ST5520_ Hipot通讯异常 *)
  通讯复位 : BOOL;
END_VAR
VAR
  判断比较字符_1 : STRING := PASS;  (* “PASS” *)
  判断比较字符_2 : STRING := LFAIL;  (* LFAIL0 *)
  判断比较字符_3 : STRING := UFAIL;  (* UFAIL0 *)
  判断比较字符_4 : STRING := ULFAIL;  (* ULFAIL *)
  判断比较字符_5 : STRING := NOCOMP;  (* NOCOMP *)
  数据空格字符 : WORD;  (* 空格 *)
  数据空格 : WORD;
  数据比较字符_2 : STRING := O.;  (* $?St$Bk?_#[574] / "O."$?St$Bk?_#[574] *)
  数据比较字符_3 : STRING := U.;  (* $?St$Bk?_#[575] / "U."$?St$Bk?_#[575] *)
  数据比较字符_4 : STRING := C.;  (* $?St$Bk?_#[576] / "C."$?St$Bk?_#[576] *)
  数据比较字符_5 : STRING := SH;  (* $?St$Bk?_#[577] / "SH"$?St$Bk?_#[577] *)
  数据比较6 : STRING := -;  (* - *)
  数据比较7 : STRING := Hi;
  数据比较8 : STRING := Ho;
  数据比较9 : STRING := HL;
  读取电阻处理_1 : STRING;
  读取电阻处理_2 : STRING;
  第一个字符 : STRING;
  Data_1 : STRING;  (* ST5520_返回绝缘测试兆欧值(String) *)
  Data_PO_2 : STRING;  (* 数据运算1（字符位置） *)
  Data_PO_3 : UINT;  (* 数据运算2（字符位置） *)
  Data_PO_4 : UINT;  (* 数据运算3（字符位置 *)
  Data_ST_5 : STRING;  (* 数据运算4（字符） *)
  Data_ST_6 : STRING;  (* 数据运算5（字符） *)
  Data_ST_7 : STRING;  (* 数据运算6（字符） *)
  COUNT_1 : UINT;  (* 复测试计数 *)
  读取判断结果_1 : STRING;
  后二个字符 : STRING;  (* 截取测试值最后一个字符 *)
  后一个字符 : STRING;
  前二个字符 : STRING;  (* 截取测试值开始二个字符 *)
  三四字符 : STRING;
  BL_1 : BOOL;  (* ST5520_A 绝缘仪读标志 *)
  BL_2 : BOOL;  (* 数据处理置位 *)
  BL_4 : BOOL;  (* 不再复测 *)
  BL_5 : BOOL;  (* 复测标志 *)
  BL : ARRAY[0..15] OF BOOL;  (* NG类型 *)
  T_1 : TIMER;  (* 读取绝缘仪延时 *)
  T_2 : TIMER;  (* 数据处理延时 *)
  T_3 : TIMER;  (* 结果判断延时 *)
  T_4 : TIMER;  (* 测试完成延时 *)
  T_5 : TIMER;  (* 复测试延时 *)
  T_6 : TIMER;  (* 断开完成延时 *)
  T_7 : TIMER;  (* 通讯报警超时 *)
  T_8 : TIMER;  (* 延时读电压 *)
  T_9 : TIMER;  (* 测试延时 *)
  BL_8 : BOOL;
  WD_3 : WORD;
  WD AT E3_32000 : ARRAY[0..199] OF WORD;
  WD1 AT E3_31000 : ARRAY[0..199] OF WORD;
  WD2 : ARRAY[0..1] OF WORD;  (* 读取电压 *)
  WD5 : STRING;
  WD6 : STRING;
  WD7 : STRING;
  WINT1 : UINT;
  WINT2 : UINT;
  WT3 : UINT;  (* 读取时间 *)
  WT4 : UINT;  (* 电压数据位 *)
  WD10 : ARRAY[0..2] OF WORD;  (* 截取数据 *)
  WD11 : ARRAY[0..2] OF WORD;  (* 截取判断结果 *)
END_VAR

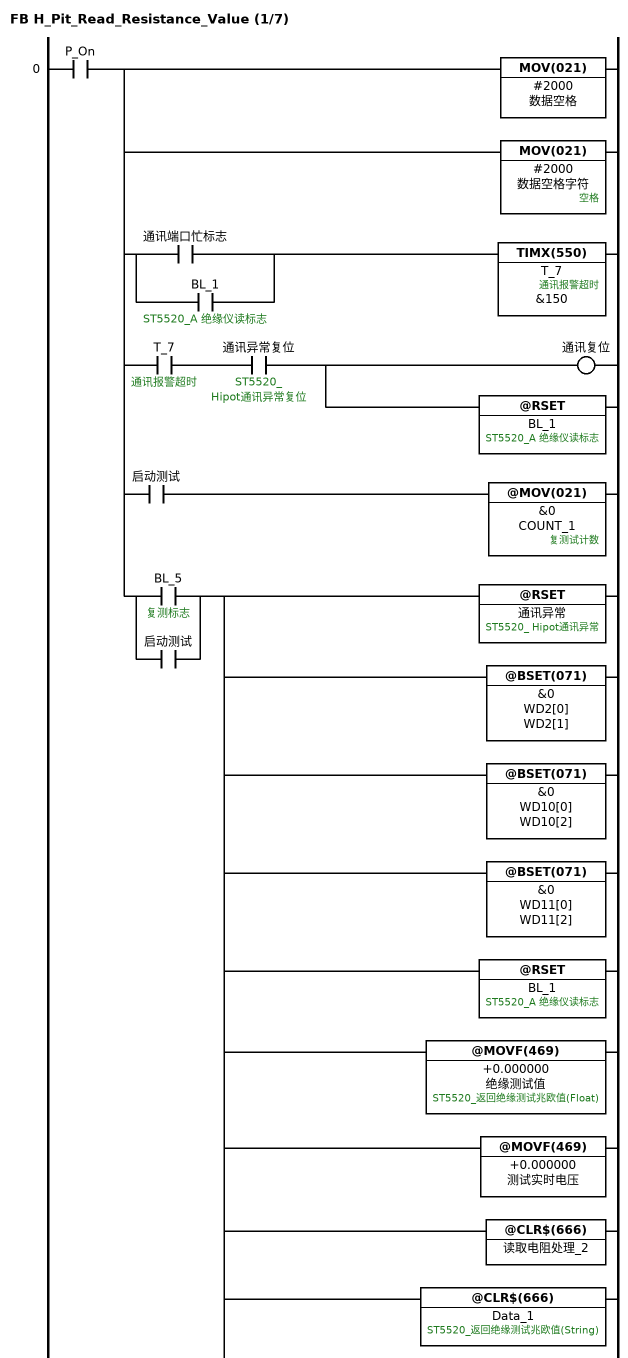

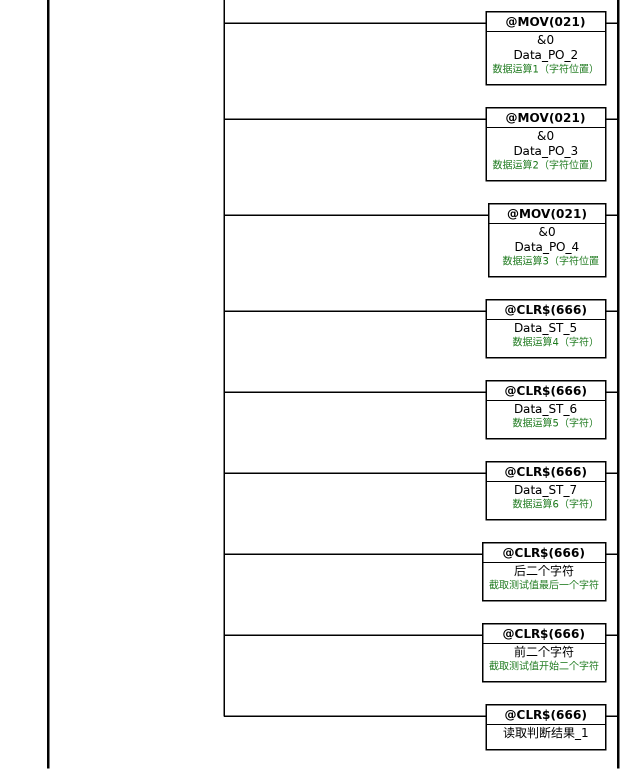
; rung 0
LD P_On
OUT TR0
MOV(021) #2000 数据空格
MOV(021) #2000 数据空格字符  ; 空格
LD 通讯端口忙标志
OR BL_1  ; ST5520_A 绝缘仪读标志
ANDLD
TIMX(550) T_7 &150  ; 通讯报警超时
LD TR0
AND T_7  ; 通讯报警超时
AND 通讯异常复位  ; ST5520_Hipot通讯异常复位
OUT 通讯复位
@RSET BL_1  ; ST5520_A 绝缘仪读标志
LD TR0
AND 启动测试
@MOV(021) &0 COUNT_1  ; 复测试计数
LD TR0
LD BL_5  ; 复测标志
OR 启动测试
ANDLD
@RSET 通讯异常  ; ST5520_ Hipot通讯异常
@BSET(071) &0 WD2[0] WD2[1]
@BSET(071) &0 WD10[0] WD10[2]
@BSET(071) &0 WD11[0] WD11[2]
@RSET BL_1  ; ST5520_A 绝缘仪读标志
@MOVF(469) +0.000000 绝缘测试值  ; ST5520_返回绝缘测试兆欧值(Float)
@MOVF(469) +0.000000 测试实时电压
@CLR$(666) 读取电阻处理_2
@CLR$(666) Data_1  ; ST5520_返回绝缘测试兆欧值(String)
@MOV(021) &0 Data_PO_2  ; 数据运算1（字符位置）
@MOV(021) &0 Data_PO_3  ; 数据运算2（字符位置）
@MOV(021) &0 Data_PO_4  ; 数据运算3（字符位置
@CLR$(666) Data_ST_5  ; 数据运算4（字符）
@CLR$(666) Data_ST_6  ; 数据运算5（字符）
@CLR$(666) Data_ST_7  ; 数据运算6（字符）
@CLR$(666) 后二个字符  ; 截取测试值最后一个字符
@CLR$(666) 前二个字符  ; 截取测试值开始二个字符
@CLR$(666) 读取判断结果_1

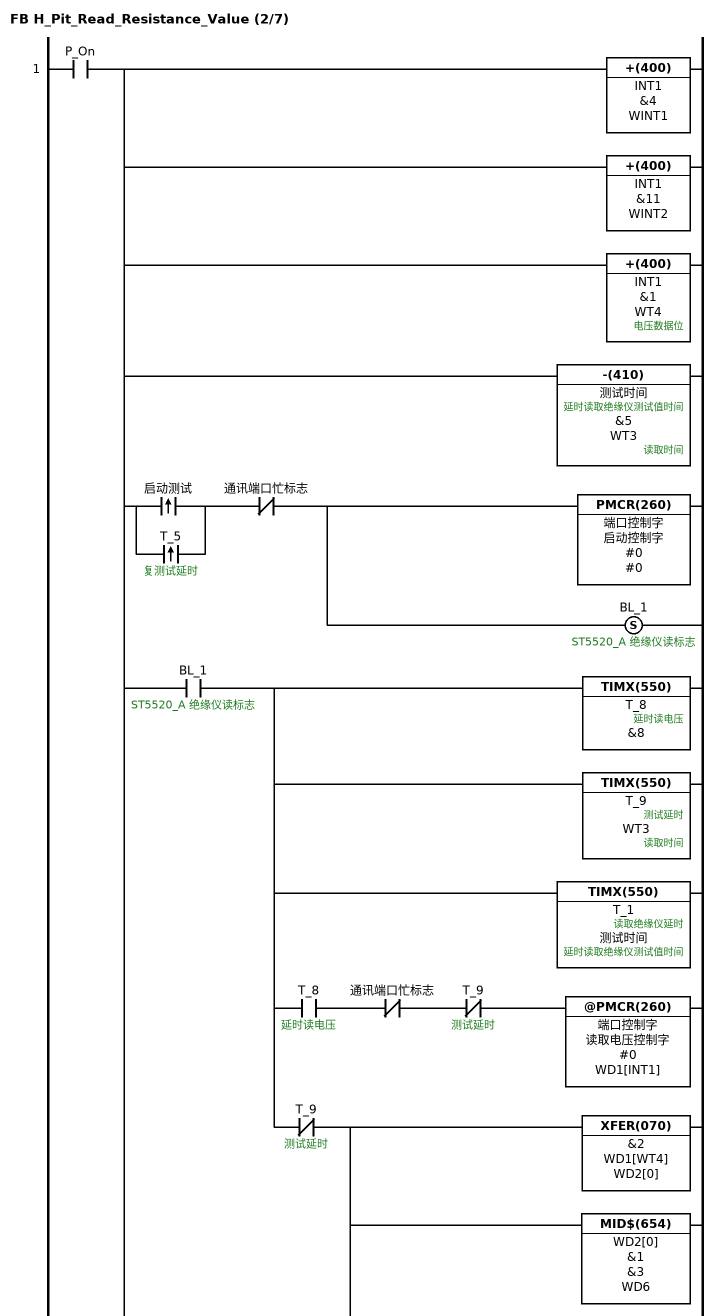

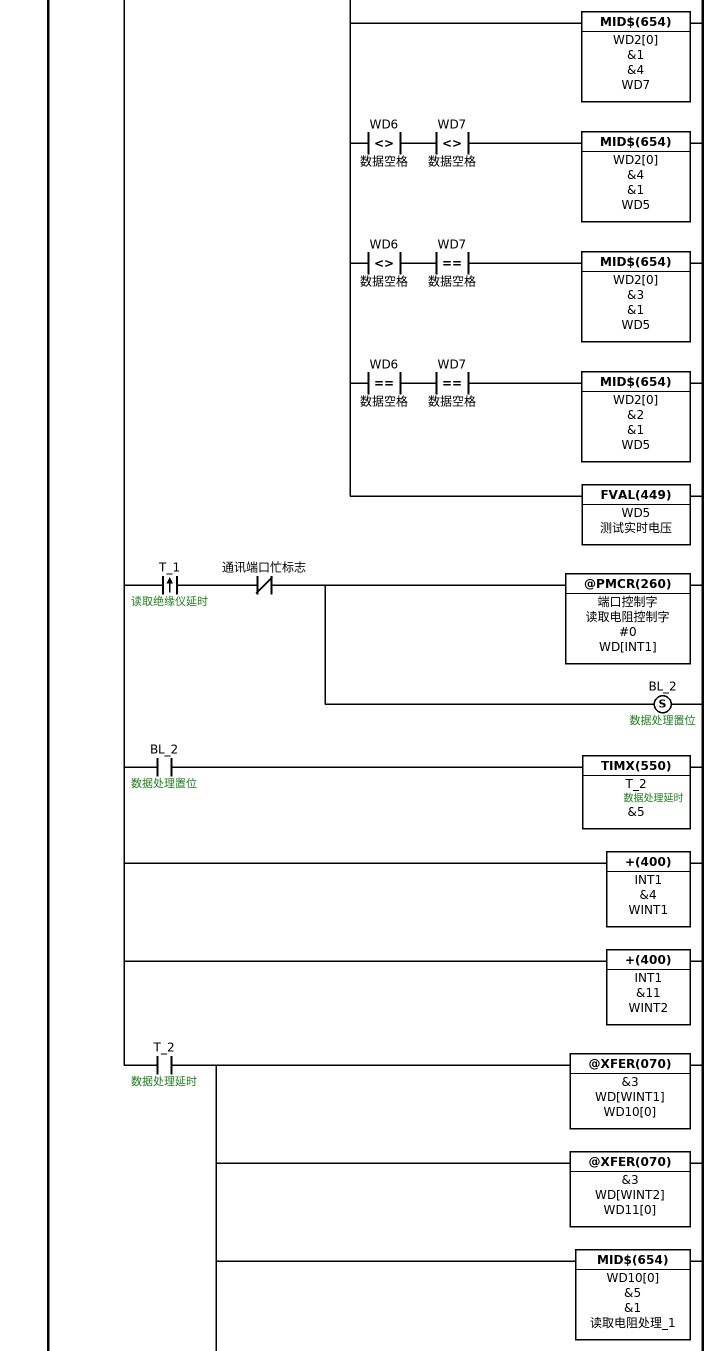

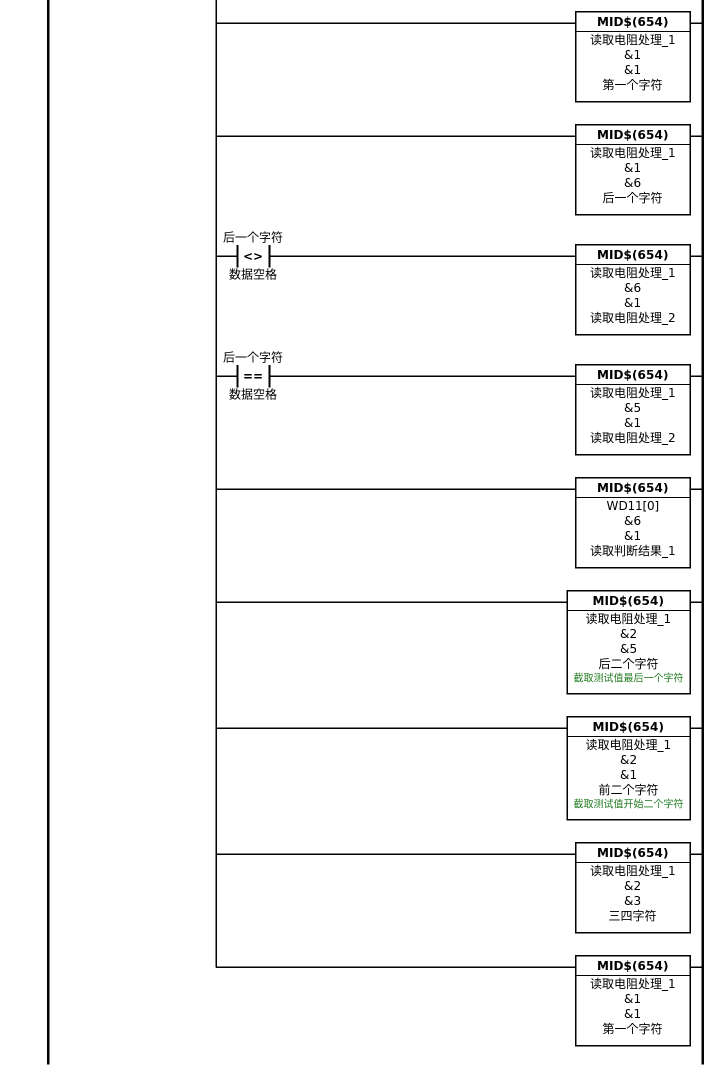
; rung 1
LD P_On
OUT TR0
+(400) INT1 &4 WINT1
+(400) INT1 &11 WINT2
+(400) INT1 &1 WT4  ; 电压数据位
-(410) 测试时间 &5 WT3  ; 延时读取绝缘仪测试值时间, 读取时间
@LD 启动测试
@OR T_5  ; 复测试延时
ANDLD
ANDNOT 通讯端口忙标志
PMCR(260) 端口控制字 启动控制字 #0 #0
SET BL_1  ; ST5520_A 绝缘仪读标志
LD TR0
AND BL_1  ; ST5520_A 绝缘仪读标志
OUT TR1
TIMX(550) T_8 &8  ; 延时读电压
TIMX(550) T_9 WT3  ; 测试延时, 读取时间
TIMX(550) T_1 测试时间  ; 读取绝缘仪延时, 延时读取绝缘仪测试值时间
AND T_8  ; 延时读电压
ANDNOT 通讯端口忙标志
ANDNOT T_9  ; 测试延时
@PMCR(260) 端口控制字 读取电压控制字 #0 WD1[INT1]
LD TR1
ANDNOT T_9  ; 测试延时
OUT TR2
XFER(070) &2 WD1[WT4] WD2[0]
MID$(654) WD2[0] &1 &3 WD6
MID$(654) WD2[0] &1 &4 WD7
AND<>(305) WD6 数据空格
AND<>(305) WD7 数据空格
MID$(654) WD2[0] &4 &1 WD5
LD TR2
AND<>(305) WD6 数据空格
AND=(300) WD7 数据空格
MID$(654) WD2[0] &3 &1 WD5
LD TR2
AND=(300) WD6 数据空格
AND=(300) WD7 数据空格
MID$(654) WD2[0] &2 &1 WD5
LD TR2
FVAL(449) WD5 测试实时电压
LD TR0
@AND T_1  ; 读取绝缘仪延时
ANDNOT 通讯端口忙标志
@PMCR(260) 端口控制字 读取电阻控制字 #0 WD[INT1]
SET BL_2  ; 数据处理置位
LD TR0
AND BL_2  ; 数据处理置位
TIMX(550) T_2 &5  ; 数据处理延时
LD TR0
+(400) INT1 &4 WINT1
+(400) INT1 &11 WINT2
AND T_2  ; 数据处理延时
OUT TR3
@XFER(070) &3 WD[WINT1] WD10[0]
@XFER(070) &3 WD[WINT2] WD11[0]
MID$(654) WD10[0] &5 &1 读取电阻处理_1
MID$(654) 读取电阻处理_1 &1 &1 第一个字符
MID$(654) 读取电阻处理_1 &1 &6 后一个字符
AND<>(305) 后一个字符 数据空格
MID$(654) 读取电阻处理_1 &6 &1 读取电阻处理_2
LD TR3
AND=(300) 后一个字符 数据空格
MID$(654) 读取电阻处理_1 &5 &1 读取电阻处理_2
LD TR3
MID$(654) WD11[0] &6 &1 读取判断结果_1
MID$(654) 读取电阻处理_1 &2 &5 后二个字符  ; 截取测试值最后一个字符
MID$(654) 读取电阻处理_1 &2 &1 前二个字符  ; 截取测试值开始二个字符
MID$(654) 读取电阻处理_1 &2 &3 三四字符
MID$(654) 读取电阻处理_1 &1 &1 第一个字符

